TYPE ST_HardSettings_Setup :
STRUCT
	//SETUP
	e_ControlSource						: eControlSources;
	
END_STRUCT
END_TYPE

(* stored: Version 1.1.0.1, ProductVersion 3.1.4026.18
   DUT ST_HardSettings_Setup: Id {142ce74d-c378-4e7d-984a-40640185cffc} *)
